TYPE ST_System_Ampel_Signal :
STRUCT
	Stellung_Rot		: BOOL;
	Stellung_Orange		: BOOL;
	Stellung_Gruen		: BOOL;
	Stellung_Blau		: BOOL;
	Stellung_Buzz		: BOOL;
END_STRUCT
END_TYPE

(* stored: Version 1.1.0.1, ProductVersion 3.1.4024.9
   DUT ST_System_Ampel_Signal: Id {86e8c406-acc9-4335-b2f5-fd3d0d692640} *)
